PROGRAM P_MachineMain
VAR
	
END_VAR

GVL_OOP.fbFeeder();
GVL_OOP.fbSTS();

END_PROGRAM

(* stored: Version 1.1.0.1, ProductVersion 3.1.4024.12
   POU P_MachineMain: Id {07331880-3efd-4696-8ef8-3d874ebc5946}, SpecialFunc None *)
